FUNCTION_BLOCK FB_Station5 EXTENDS FB_PackML_BaseModule
VAR
	VirtualOffsetMasterAxis : FB_Component_BasicAxis	  := (Name := 'Station 5 Virtual Offset Master Axis');
	VirtualCammedMasterAxis : FB_Component_CamSlaveAxis	  := (Name := 'Station 5 Virtual Cam Axis');
	CammedOffsetAxis		: FB_Component_BasicSlaveAxis := (Name := 'Station 5 Cammed Offset Axis');
	_MasterRef				: REFERENCE TO AXIS_REF;
	CamParameters			: ST_CamParameters;
	V_OffsetFWD				: BOOL;
	V_OffsetREV				: BOOL;
END_VAR

(*
	Design Considerations:
		Why use a Virtual Axis?
			Software/Virtual axes can be easily managed from within TwinCAT PLC and NC. 
			Notably the encoder value can be changed without physical movement and with no impact to real hardware.
			Therefore, it is possible to set position on a virtual axis to a specific value without physical movement an with no impact to the coupled axis.

			When using a Virtual axis for a Cam table, the real axis can be decoupled, 
			then the virtual cam table slave can be adjusted as needed, and then the real axis can couple to the virtual axis.
						
	
	Components:
		VirtualOffsetMasterAxis - Local virtual axis used to apply an offset to the real axis position
		VirtualCammedMasterAxis - follows the cam table with the MachineVirtualAxis as the master axis of the table.
			The Cam table is a move from 0 - 100
		CammedOffsetAxis - geared to the VirtualCammedMasterAxis and the VirtualCammedMasterAxis, and will follow commands from both.

	Methods:
		CyclicLogic - 
			Monitors the HMI variables to move the VirtualOffsetMasterAxis +/- 100
			
		Initialize - 
			Create the Cam table data and set the Component (VirtualCammedMasterAxis) CamParameters Ref to the data after the component is initialized
			Set the Component (VirtualCammedMasterAxis) Master axis Ref to the Property backer variable for _MasterAxisRef after the component is initialized
			Set the Component (CammedOffsetAxis) Master1 axis Ref to the Component (VirtualCammedMasterAxis) Axis property after the component is initialized
			Set the Component (CammedOffsetAxis) Master2 axis Ref to the Component (VirtualOffsetMasterAxis) Axis property after the component is initialized
	
	
		Starting - 
			Calls StartSync method of VirtualCammedMasterAxis to cam axis to table
			Couples the CammedOffsetAxis to both master axes		
			
*)

METHOD PROTECTED Aborting
//Mode is ignored
CASE SequenceState OF
	0:
		NoStateTasksToComplete := FALSE;
		SequenceState		   := SequenceState + 10;

	10: (* Stop Axis *)

		//Setting Override to 100 will ensure velocity calculations are not limited
		VirtualOffsetMasterAxis.Override := 100;
		VirtualCammedMasterAxis.Override := 100;
		CammedOffsetAxis.Override		 := 100;

		//
		IF VirtualOffsetMasterAxis.Stop() THEN //This will also GearOut by default
			SequenceState := SequenceState + 10;
		END_IF

	20:
		IF VirtualCammedMasterAxis.Stop() THEN //This will also GearOut by default
			SequenceState := SequenceState + 10;
		END_IF

	30:
		IF CammedOffsetAxis.Stop() THEN //This will also GearOut by default
			SequenceState := SequenceState + 10;
		END_IF

	40:
		IF VirtualOffsetMasterAxis.Stopped AND VirtualCammedMasterAxis.Stopped AND CammedOffsetAxis.Stopped THEN
			SequenceState := SequenceState + 10;
		END_IF

	50: (* Disable Axis *)
		IF VirtualOffsetMasterAxis.Disable() THEN
			SequenceState := SequenceState + 10;
		END_IF

	60: (* Disable Axis *)
		IF VirtualCammedMasterAxis.Disable() THEN
			SequenceState := SequenceState + 10;
		END_IF

	70: (* Disable Axis *)
		IF CammedOffsetAxis.Disable() THEN
			SequenceState := SequenceState + 10;
		END_IF

	80:
		IF NOT VirtualOffsetMasterAxis.Enabled AND NOT VirtualCammedMasterAxis.Enabled AND NOT CammedOffsetAxis.Enabled THEN
			SequenceState := SequenceState + 10;
		END_IF

	90:
		StateTasksComplete := TRUE;
END_CASE

SUPER^.Aborting();
END_METHOD

METHOD PROTECTED Completing
CASE SequenceState OF
	0:
		NoStateTasksToComplete := FALSE;
		SequenceState		   := SequenceState + 10;

	10:
		IF VirtualOffsetMasterAxis.Stop() THEN //This will also GearOut
			SequenceState := SequenceState + 10;
		END_IF

	20:
		IF VirtualCammedMasterAxis.Stop() THEN //This will also GearOut
			SequenceState := SequenceState + 10;
		END_IF

	30:
		IF CammedOffsetAxis.Stop() THEN //This will also GearOut
			SequenceState := SequenceState + 10;
		END_IF

	40:
		IF VirtualOffsetMasterAxis.Stopped AND VirtualCammedMasterAxis.Stopped AND CammedOffsetAxis.Stopped THEN
			SequenceState := SequenceState + 10;
		END_IF

	50:
		StateTasksComplete := TRUE;
END_CASE

SUPER^.Completing();
END_METHOD

METHOD PUBLIC CyclicLogic
IF NOT InitComplete THEN
	_InitComplete := Initialize();
	RETURN;
END_IF

//Move commands from Visu
IF V_OffsetFWD THEN
	VirtualOffsetMasterAxis.MoveRelative(100, 0);
END_IF

IF V_OffsetREV THEN
	VirtualOffsetMasterAxis.MoveRelative(-100, 0);
END_IF

//
SUPER^.CyclicLogic();
END_METHOD

METHOD PROTECTED Initialize : BOOL;
Initialize := FALSE;
CASE DescendantSequenceState OF
	0:
		RegisterComponent(VirtualOffsetMasterAxis);
		RegisterComponent(VirtualCammedMasterAxis);
		RegisterComponent(CammedOffsetAxis);
		DescendantSequenceState := DescendantSequenceState + 10;

	10:
		IF SUPER^.Initialize() THEN
			//Create the Cam table data and set the Component (VirtualCammedMasterAxis) CamParameters Ref to the data after the component is initialized
			WriteCamParameters();
			VirtualCammedMasterAxis.CamParameters REF= CamParameters;

			//Setting the Reference of the FB_Component_CamSlaveAxis must be done after the component has been initialized
			VirtualCammedMasterAxis.Master REF= _MasterRef;

			//Setting the Reference of the FB_Component_BasicSlaveAxis must be done after the component has been initialized
			CammedOffsetAxis.Master1 REF= VirtualCammedMasterAxis.Axis;
			CammedOffsetAxis.Master2 REF= VirtualOffsetMasterAxis.Axis;

			//
			DescendantSequenceState := DescendantSequenceState + 10;
		END_IF

	20:
		Initialize := TRUE;
END_CASE
END_METHOD

PROPERTY MasterAxisRef : REFERENCE TO AXIS_REF
SET
_MasterRef REF= MasterAxisRef;
END_SET
END_PROPERTY

METHOD PROTECTED Starting
CASE _CommandedMode OF
	ePMLProtUnitMode_Production:
		CASE SequenceState OF
			0:
				NoStateTasksToComplete := FALSE;
				SequenceState		   := SequenceState + 10;

			10: (* Enable Axis *)
				IF VirtualCammedMasterAxis.Enable() THEN
					SequenceState := SequenceState + 10;
				END_IF

			20:
				IF VirtualCammedMasterAxis.Enabled THEN
					SequenceState := SequenceState + 10;
				END_IF

			30:
				IF VirtualCammedMasterAxis.MoveAbsolute(0, 0) THEN
					SequenceState := SequenceState + 10;
				END_IF

			40:
				IF NOT VirtualCammedMasterAxis.Busy THEN
					IF NOT VirtualCammedMasterAxis.Error THEN
						SequenceState := SequenceState + 10;
					END_IF
				END_IF

			50: (* Enable Axis *)
				IF VirtualOffsetMasterAxis.Enable() THEN
					SequenceState := SequenceState + 10;
				END_IF

			60:
				IF VirtualOffsetMasterAxis.Enabled THEN
					SequenceState := SequenceState + 10;
				END_IF

			70:
				IF VirtualOffsetMasterAxis.MoveAbsolute(0, 0) THEN
					SequenceState := SequenceState + 10;
				END_IF

			80:
				IF NOT VirtualOffsetMasterAxis.Busy THEN
					IF NOT VirtualOffsetMasterAxis.Error THEN
						SequenceState := SequenceState + 10;
					END_IF
				END_IF

			90: (* Verify the Master axis is ready *)
				IF VirtualCammedMasterAxis.Master.Status.Operational THEN
					IF VirtualCammedMasterAxis.Master.NcToPlc.ActPos = 0.0 THEN
						SequenceState := SequenceState + 10;
					END_IF
				END_IF

			100: (* Couple to Cam table with Master axis*)
				IF VirtualCammedMasterAxis.StartSync() THEN
					SequenceState := SequenceState + 10;
				END_IF

			110:
				IF VirtualCammedMasterAxis.InSync THEN
					SequenceState := SequenceState + 10;
				END_IF

			120: (* Enable Axis *)
				IF CammedOffsetAxis.Enable() THEN
					SequenceState := SequenceState + 10;
				END_IF

			130:
				IF CammedOffsetAxis.Enabled THEN
					SequenceState := SequenceState + 10;
				END_IF

			140:
				IF CammedOffsetAxis.MoveAbsolute(0, 0) THEN
					SequenceState := SequenceState + 10;
				END_IF

			150:
				IF NOT CammedOffsetAxis.Busy THEN
					IF NOT CammedOffsetAxis.Error THEN
						SequenceState := SequenceState + 10;
					END_IF
				END_IF

			160: (* Verify the Master axis is ready *)
				IF CammedOffsetAxis.Master1.Status.Operational THEN
					//A small tolerance of position is used becaused the Axis moves by a small amount when cammed in 
					IF CammedOffsetAxis.Master1.NcToPlc.ActPos <= 0.01 AND CammedOffsetAxis.Master1.NcToPlc.ActPos >= -0.01 THEN
						SequenceState := SequenceState + 10;
					END_IF
				END_IF

			170: (* Couple to Master axis *)
				IF CammedOffsetAxis.GearIn() THEN
					SequenceState := SequenceState + 10;
				END_IF

			180:
				IF CammedOffsetAxis.InGear THEN
					SequenceState := SequenceState + 10;
				END_IF

			190:
				StateTasksComplete := TRUE;
		END_CASE
END_CASE

SUPER^.Starting();
END_METHOD

METHOD PROTECTED Stopping
CASE SequenceState OF
	0:
		NoStateTasksToComplete := FALSE;
		SequenceState		   := SequenceState + 10;

	10:
		IF VirtualOffsetMasterAxis.Stop() THEN //This will also GearOut by default
			SequenceState := SequenceState + 10;
		END_IF

	20:
		IF VirtualCammedMasterAxis.Stop() THEN //This will also GearOut by default
			SequenceState := SequenceState + 10;
		END_IF

	30:
		IF CammedOffsetAxis.Stop() THEN //This will also GearOut by default
			SequenceState := SequenceState + 10;
		END_IF

	40:
		IF VirtualOffsetMasterAxis.Stopped AND VirtualCammedMasterAxis.Stopped AND CammedOffsetAxis.Stopped THEN
			SequenceState := SequenceState + 10;
		END_IF

	50:
		StateTasksComplete := TRUE;
END_CASE

SUPER^.Stopping();
END_METHOD

METHOD WriteCamParameters
CamParameters.CamTableId := VirtualCammedMasterAxis.Axis.NcToPlc.AxisId;

//Table 1
CamParameters.CamTable[1].NumberOfPoints			  := 3;
CamParameters.CamTable[1].Points[1].PointIndex		  := 1;
CamParameters.CamTable[1].Points[1].FunctionType	  := MC_MotionFunctionType.MOTIONFUNCTYPE_POLYNOM5;
CamParameters.CamTable[1].Points[1].PointType		  := MC_MotionPointType.MOTIONPOINTTYPE_REST;
CamParameters.CamTable[1].Points[1].RelIndexNextPoint := 1;
CamParameters.CamTable[1].Points[1].MasterPos		  := 0.0;
CamParameters.CamTable[1].Points[1].SlavePos		  := 0.0;
CamParameters.CamTable[1].Points[2].PointIndex		  := 2;
CamParameters.CamTable[1].Points[2].FunctionType	  := MC_MotionFunctionType.MOTIONFUNCTYPE_POLYNOM5;
CamParameters.CamTable[1].Points[2].PointType		  := MC_MotionPointType.MOTIONPOINTTYPE_TURN;
CamParameters.CamTable[1].Points[2].RelIndexNextPoint := 1;
CamParameters.CamTable[1].Points[2].MasterPos		  := 180.0;
CamParameters.CamTable[1].Points[2].SlavePos		  := 100.0;
CamParameters.CamTable[1].Points[3].PointIndex		  := 3;
CamParameters.CamTable[1].Points[3].FunctionType	  := MC_MotionFunctionType.MOTIONFUNCTYPE_POLYNOM5;
CamParameters.CamTable[1].Points[3].PointType		  := MC_MotionPointType.MOTIONPOINTTYPE_REST;
CamParameters.CamTable[1].Points[3].RelIndexNextPoint := 0;
CamParameters.CamTable[1].Points[3].MasterPos		  := 360.0;
CamParameters.CamTable[1].Points[3].SlavePos		  := 0.0;
CamParameters.CamTable[1].NumberOfPoints			  := 3;
END_METHOD

END_FUNCTION_BLOCK

(* stored: Version 1.1.0.1, ProductVersion 3.1.4024.12
   POU FB_Station5: Id {26b1d8bf-573e-4474-9908-1cb3f660443a}, SpecialFunc None
   Folder Acting States: Id {33bd8a36-e5b1-4365-a662-b02628e2a824}
   Folder I_CyclicFB: Id {2980bb69-ab02-4bfb-ad1c-9fa03d9a2716}
   Folder Methods: Id {3c4bbf80-232f-47ea-b70f-1909e0d359ef}
   Folder Properties: Id {256e166a-44bc-4ff6-9c38-8298e3837af6}
   Method Aborting: Id {19f60301-d4a8-4792-8221-bddbaf6a02dc}
   Method Completing: Id {69befc6a-34d8-463e-ac5c-da3822eced32}
   Method CyclicLogic: Id {02ff2b48-1baf-493b-bd66-c94f3e23bfb8}
   Method Initialize: Id {9402b14e-f209-4168-b1e3-2b85ca890ad5}
   Property MasterAxisRef: Id {27d2aaee-04b1-4a43-af5b-2a694b8e7aee}
   Set Set: Id {4cf51866-b61c-4187-b337-138cbd2df373}
   Method Starting: Id {62bd265c-6ee7-4c9c-860a-ad4e286fb110}
   Method Stopping: Id {87f49bba-e9a6-4150-ad57-c615728b1634}
   Method WriteCamParameters: Id {a73be485-93b9-4d7c-9010-73a79c5946b4} *)
